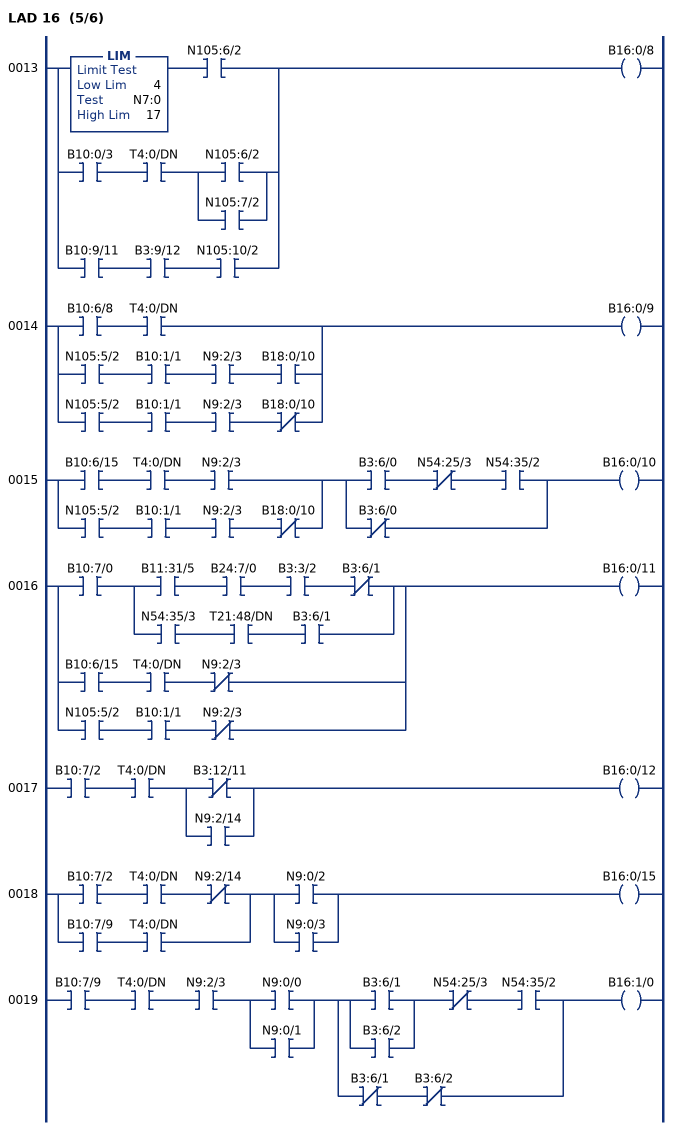
% Rung: 13 %
SOR BST LIM 4 N7:0 17 XIC N105:6/2 NXB XIC B10:0/3 XIC T4:0/DN BST XIC N105:6/2 NXB XIC N105:7/2 BND NXB XIC B10:9/11 XIC B3:9/12 XIC N105:10/2 BND OTE B16:0/8 EOR
% Rung: 14 %
SOR BST XIC B10:6/8 XIC T4:0/DN NXB XIC N105:5/2 XIC B10:1/1 XIC N9:2/3 XIC B18:0/10 NXB XIC N105:5/2 XIC B10:1/1 XIC N9:2/3 XIO B18:0/10 BND OTE B16:0/9 EOR
% Rung: 15 %
SOR BST XIC B10:6/15 XIC T4:0/DN XIC N9:2/3 NXB XIC N105:5/2 XIC B10:1/1 XIC N9:2/3 XIO B18:0/10 BND BST XIC B3:6/0 XIO N54:25/3 XIC N54:35/2 NXB XIO B3:6/0 BND OTE B16:0/10 EOR
% Rung: 16 %
SOR BST BST XIC B10:7/0 BST XIC B11:31/5 XIC B24:7/0 XIC B3:3/2 XIO B3:6/1 NXB XIC N54:35/3 XIC T21:48/DN XIC B3:6/1 BND NXB XIC B10:6/15 XIC T4:0/DN XIO N9:2/3 BND NXB XIC N105:5/2 XIC B10:1/1 XIO N9:2/3 BND OTE B16:0/11 EOR
% Rung: 17 %
SOR XIC B10:7/2 XIC T4:0/DN BST XIO B3:12/11 NXB XIC N9:2/14 BND OTE B16:0/12 EOR
% Rung: 18 %
SOR BST XIC B10:7/2 XIC T4:0/DN XIO N9:2/14 NXB XIC B10:7/9 XIC T4:0/DN BND BST XIC N9:0/2 NXB XIC N9:0/3 BND OTE B16:0/15 EOR
% Rung: 19 %
SOR XIC B10:7/9 XIC T4:0/DN XIC N9:2/3 BST XIC N9:0/0 NXB XIC N9:0/1 BND BST BST XIC B3:6/1 NXB XIC B3:6/2 BND XIO N54:25/3 XIC N54:35/2 NXB XIO B3:6/1 XIO B3:6/2 BND OTE B16:1/0 EOR

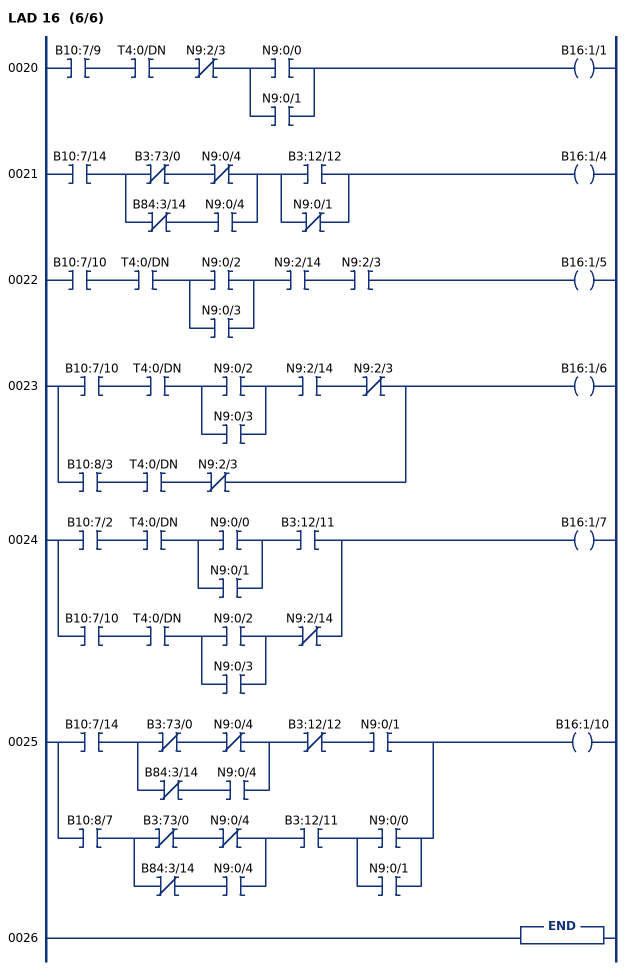
% Rung: 20 %
SOR XIC B10:7/9 XIC T4:0/DN XIO N9:2/3 BST XIC N9:0/0 NXB XIC N9:0/1 BND OTE B16:1/1 EOR
% Rung: 21 %
SOR XIC B10:7/14 BST XIO B3:73/0 XIO N9:0/4 NXB XIO B84:3/14 XIC N9:0/4 BND BST XIC B3:12/12 NXB XIO N9:0/1 BND OTE B16:1/4 EOR
% Rung: 22 %
SOR XIC B10:7/10 XIC T4:0/DN BST XIC N9:0/2 NXB XIC N9:0/3 BND XIC N9:2/14 XIC N9:2/3 OTE B16:1/5 EOR
% Rung: 23 %
SOR BST XIC B10:7/10 XIC T4:0/DN BST XIC N9:0/2 NXB XIC N9:0/3 BND XIC N9:2/14 XIO N9:2/3 NXB XIC B10:8/3 XIC T4:0/DN XIO N9:2/3 BND OTE B16:1/6 EOR
% Rung: 24 %
SOR BST XIC B10:7/2 XIC T4:0/DN BST XIC N9:0/0 NXB XIC N9:0/1 BND XIC B3:12/11 NXB XIC B10:7/10 XIC T4:0/DN BST XIC N9:0/2 NXB XIC N9:0/3 BND XIO N9:2/14 BND OTE B16:1/7 EOR
% Rung: 25 %
SOR BST XIC B10:7/14 BST XIO B3:73/0 XIO N9:0/4 NXB XIO B84:3/14 XIC N9:0/4 BND XIO B3:12/12 XIC N9:0/1 NXB XIC B10:8/7 BST XIO B3:73/0 XIO N9:0/4 NXB XIO B84:3/14 XIC N9:0/4 BND XIC B3:12/11 BST XIC N9:0/0 NXB XIC N9:0/1 BND BND OTE B16:1/10 EOR
% Rung: 26 %
SOR END EOR

LADDER 17
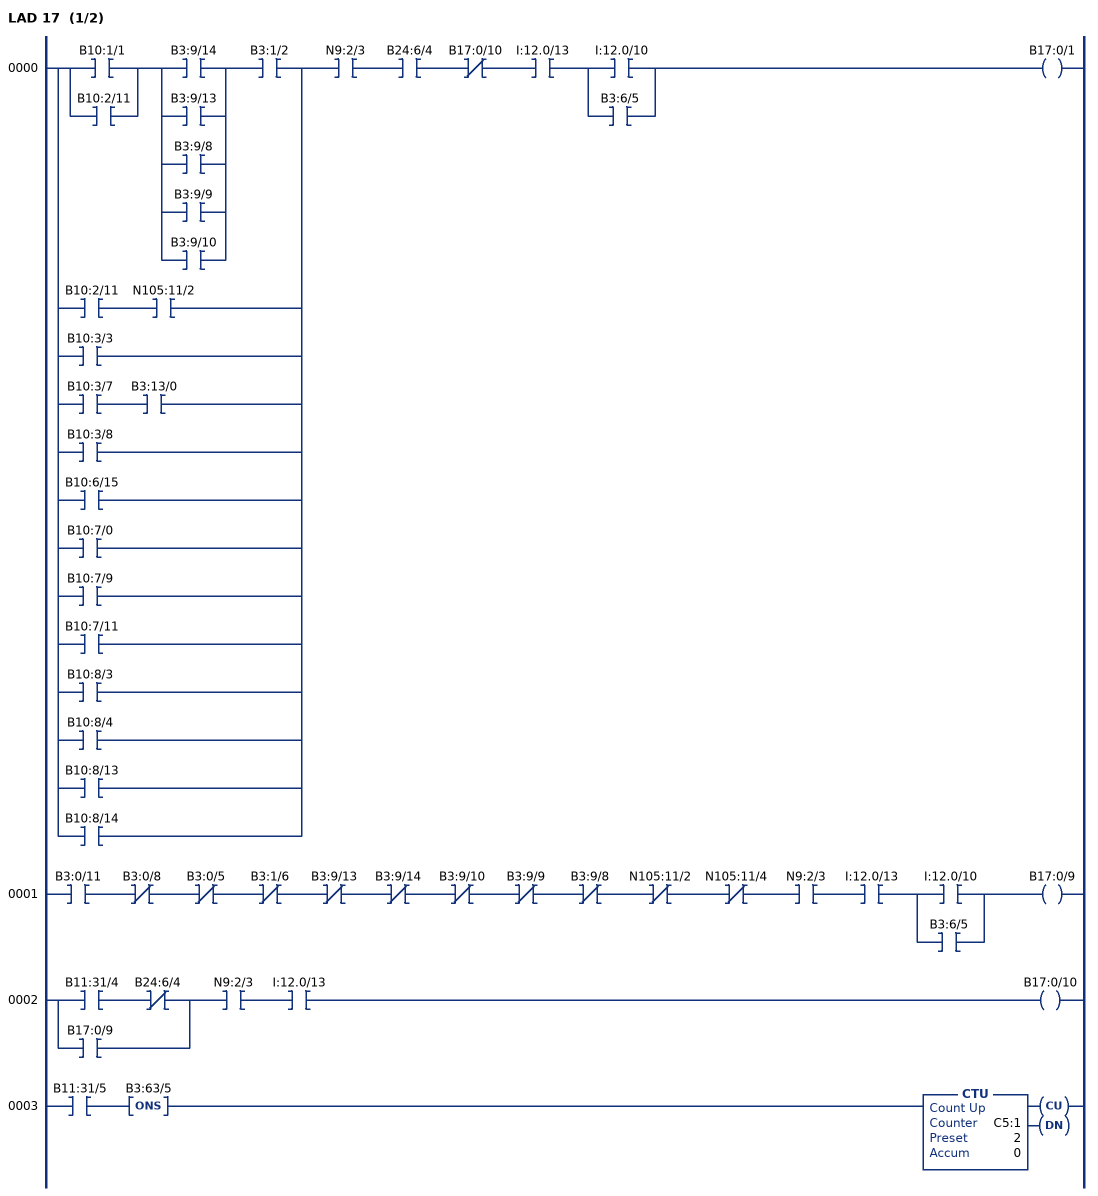
% Rung: 0 %
SOR BST BST XIC B10:1/1 NXB XIC B10:2/11 BND BST XIC B3:9/14 NXB XIC B3:9/13 NXB XIC B3:9/8 NXB XIC B3:9/9 NXB XIC B3:9/10 BND XIC B3:1/2 NXB XIC B10:2/11 XIC N105:11/2 NXB XIC B10:3/3 NXB XIC B10:3/7 XIC B3:13/0 NXB XIC B10:3/8 NXB XIC B10:6/15 NXB XIC B10:7/0 NXB XIC B10:7/9 NXB XIC B10:7/11 NXB XIC B10:8/3 NXB XIC B10:8/4 NXB XIC B10:8/13 NXB XIC B10:8/14 BND XIC N9:2/3 XIC B24:6/4 XIO B17:0/10 XIC I:12.0/13 BST XIC I:12.0/10 NXB XIC B3:6/5 BND OTE B17:0/1 EOR
% Rung: 1 %
SOR XIC B3:0/11 XIO B3:0/8 XIO B3:0/5 XIO B3:1/6 XIO B3:9/13 XIO B3:9/14 XIO B3:9/10 XIO B3:9/9 XIO B3:9/8 XIO N105:11/2 XIO N105:11/4 XIC N9:2/3 XIC I:12.0/13 BST XIC I:12.0/10 NXB XIC B3:6/5 BND OTE B17:0/9 EOR
% Rung: 2 %
SOR BST XIC B11:31/4 XIO B24:6/4 NXB XIC B17:0/9 BND XIC N9:2/3 XIC I:12.0/13 OTE B17:0/10 EOR
% Rung: 3 %
SOR XIC B11:31/5 OSR B3:63/5 CTU C5:1 2 0 EOR

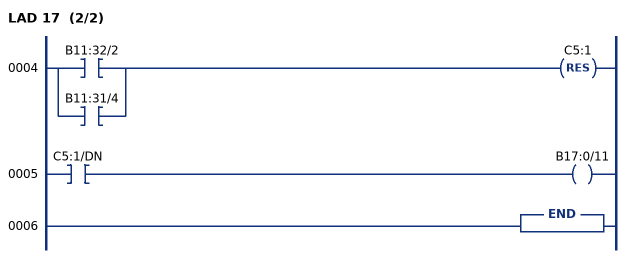
% Rung: 4 %
SOR BST XIC B11:32/2 NXB XIC B11:31/4 BND RES C5:1 EOR
% Rung: 5 %
SOR XIC C5:1/DN OTE B17:0/11 EOR
% Rung: 6 %
SOR END EOR

LADDER 18
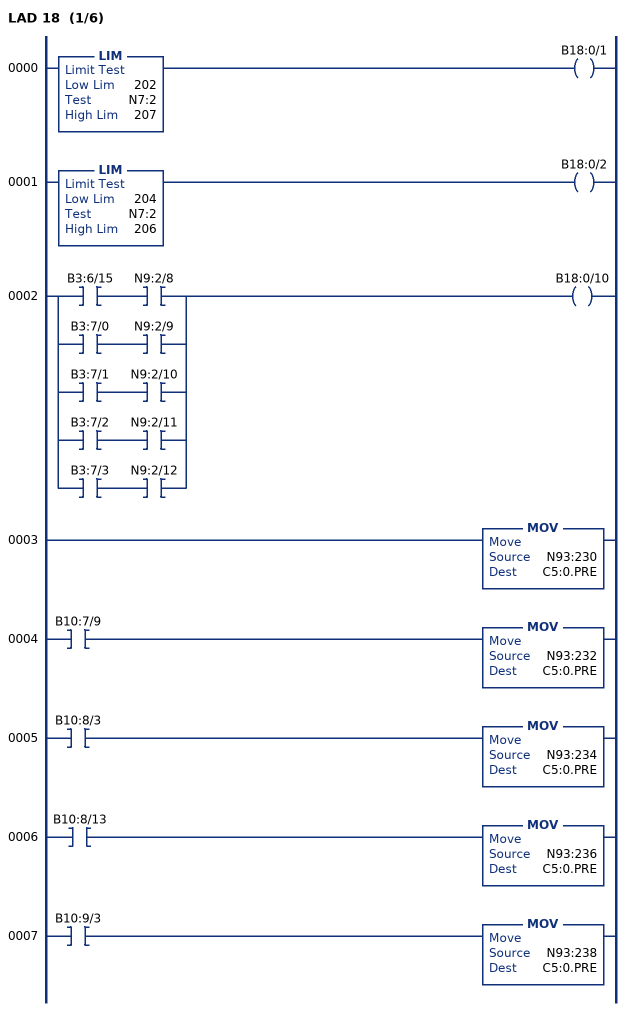
% Rung: 0 %
SOR LIM 202 N7:2 207 OTE B18:0/1 EOR
% Rung: 1 %
SOR LIM 204 N7:2 206 OTE B18:0/2 EOR
% Rung: 2 %
SOR BST XIC B3:6/15 XIC N9:2/8 NXB XIC B3:7/0 XIC N9:2/9 NXB XIC B3:7/1 XIC N9:2/10 NXB XIC B3:7/2 XIC N9:2/11 NXB XIC B3:7/3 XIC N9:2/12 BND OTE B18:0/10 EOR
% Rung: 3 %
SOR MOV N93:230 C5:0.PRE EOR
% Rung: 4 %
SOR XIC B10:7/9 MOV N93:232 C5:0.PRE EOR
% Rung: 5 %
SOR XIC B10:8/3 MOV N93:234 C5:0.PRE EOR
% Rung: 6 %
SOR XIC B10:8/13 MOV N93:236 C5:0.PRE EOR
% Rung: 7 %
SOR XIC B10:9/3 MOV N93:238 C5:0.PRE EOR

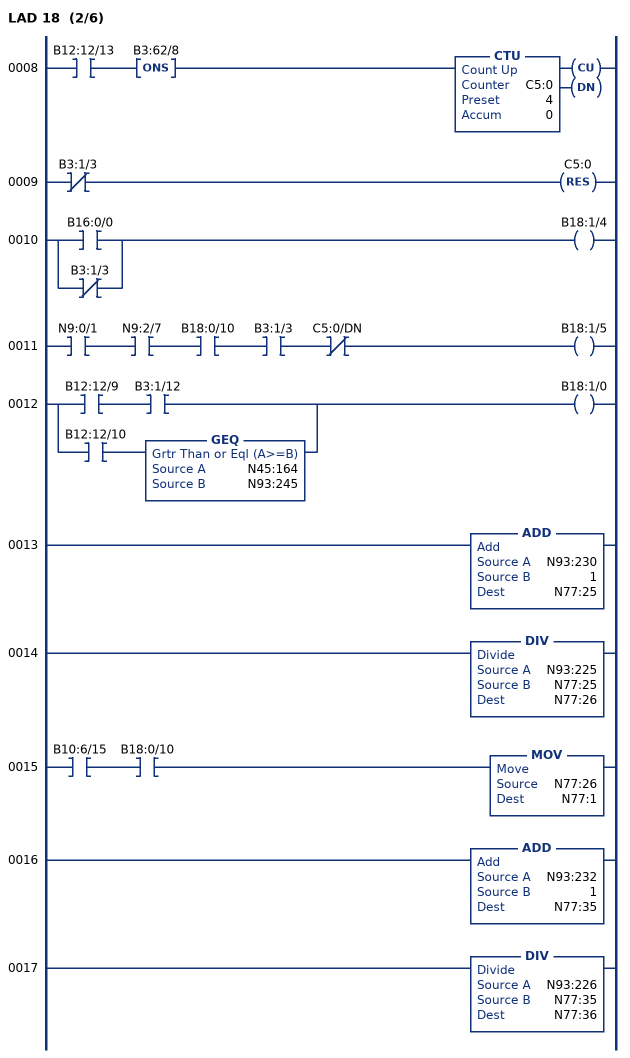
% Rung: 8 %
SOR XIC B12:12/13 OSR B3:62/8 CTU C5:0 4 0 EOR
% Rung: 9 %
SOR XIO B3:1/3 RES C5:0 EOR
% Rung: 10 %
SOR BST XIC B16:0/0 NXB XIO B3:1/3 BND OTE B18:1/4 EOR
% Rung: 11 %
SOR XIC N9:0/1 XIC N9:2/7 XIC B18:0/10 XIC B3:1/3 XIO C5:0/DN OTE B18:1/5 EOR
% Rung: 12 %
SOR BST XIC B12:12/9 XIC B3:1/12 NXB XIC B12:12/10 GEQ N45:164 N93:245 BND OTE B18:1/0 EOR
% Rung: 13 %
SOR ADD N93:230 1 N77:25 EOR
% Rung: 14 %
SOR DIV N93:225 N77:25 N77:26 EOR
% Rung: 15 %
SOR XIC B10:6/15 XIC B18:0/10 MOV N77:26 N77:1 EOR
% Rung: 16 %
SOR ADD N93:232 1 N77:35 EOR
% Rung: 17 %
SOR DIV N93:226 N77:35 N77:36 EOR

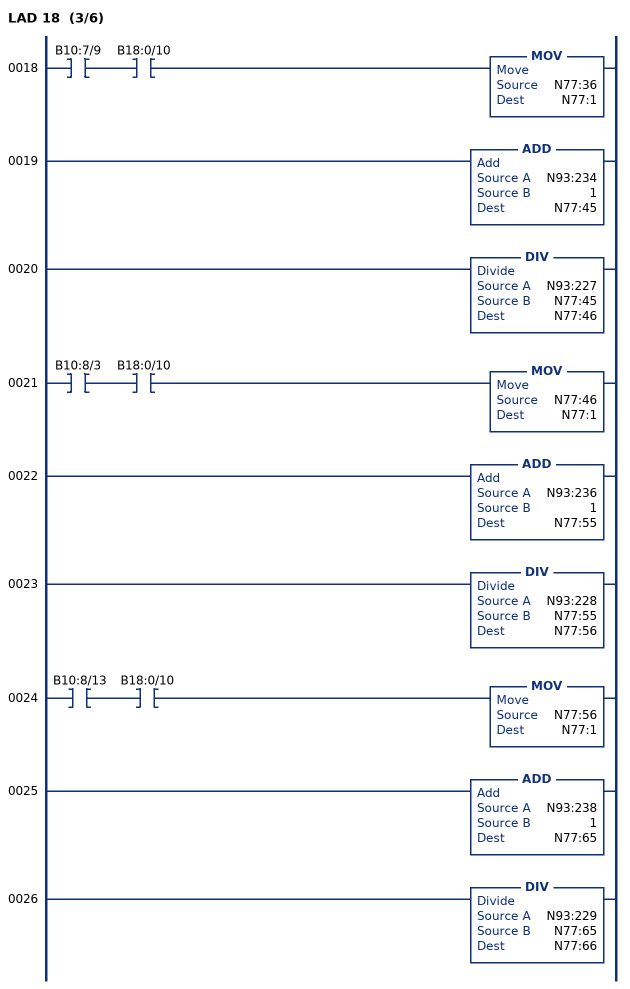
% Rung: 18 %
SOR XIC B10:7/9 XIC B18:0/10 MOV N77:36 N77:1 EOR
% Rung: 19 %
SOR ADD N93:234 1 N77:45 EOR
% Rung: 20 %
SOR DIV N93:227 N77:45 N77:46 EOR
% Rung: 21 %
SOR XIC B10:8/3 XIC B18:0/10 MOV N77:46 N77:1 EOR
% Rung: 22 %
SOR ADD N93:236 1 N77:55 EOR
% Rung: 23 %
SOR DIV N93:228 N77:55 N77:56 EOR
% Rung: 24 %
SOR XIC B10:8/13 XIC B18:0/10 MOV N77:56 N77:1 EOR
% Rung: 25 %
SOR ADD N93:238 1 N77:65 EOR
% Rung: 26 %
SOR DIV N93:229 N77:65 N77:66 EOR

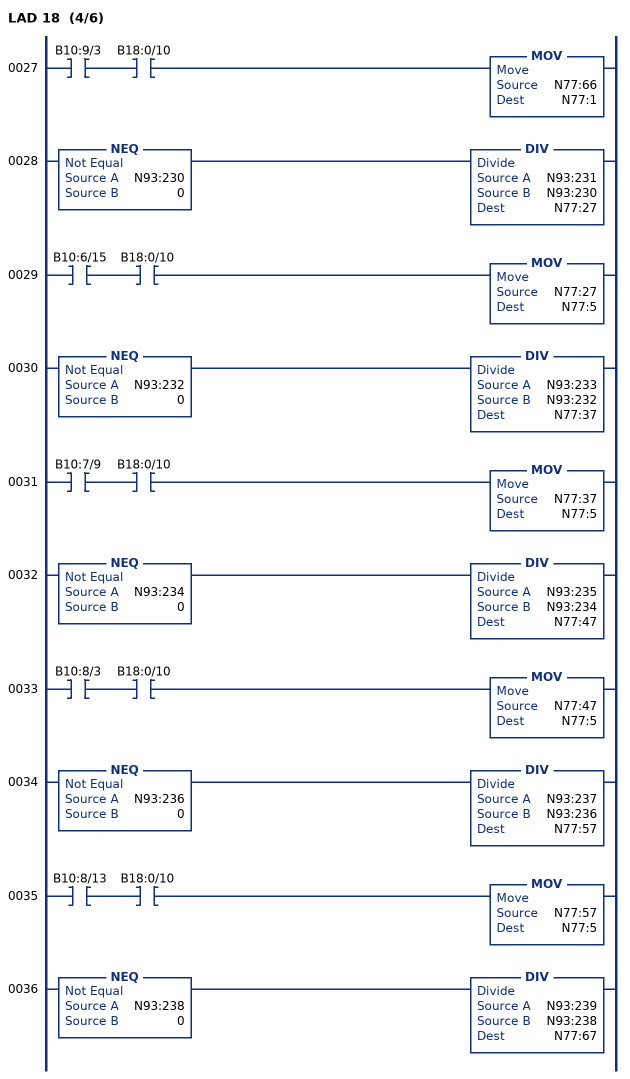
% Rung: 27 %
SOR XIC B10:9/3 XIC B18:0/10 MOV N77:66 N77:1 EOR
% Rung: 28 %
SOR NEQ N93:230 0 DIV N93:231 N93:230 N77:27 EOR
% Rung: 29 %
SOR XIC B10:6/15 XIC B18:0/10 MOV N77:27 N77:5 EOR
% Rung: 30 %
SOR NEQ N93:232 0 DIV N93:233 N93:232 N77:37 EOR
% Rung: 31 %
SOR XIC B10:7/9 XIC B18:0/10 MOV N77:37 N77:5 EOR
% Rung: 32 %
SOR NEQ N93:234 0 DIV N93:235 N93:234 N77:47 EOR
% Rung: 33 %
SOR XIC B10:8/3 XIC B18:0/10 MOV N77:47 N77:5 EOR
% Rung: 34 %
SOR NEQ N93:236 0 DIV N93:237 N93:236 N77:57 EOR
% Rung: 35 %
SOR XIC B10:8/13 XIC B18:0/10 MOV N77:57 N77:5 EOR
% Rung: 36 %
SOR NEQ N93:238 0 DIV N93:239 N93:238 N77:67 EOR

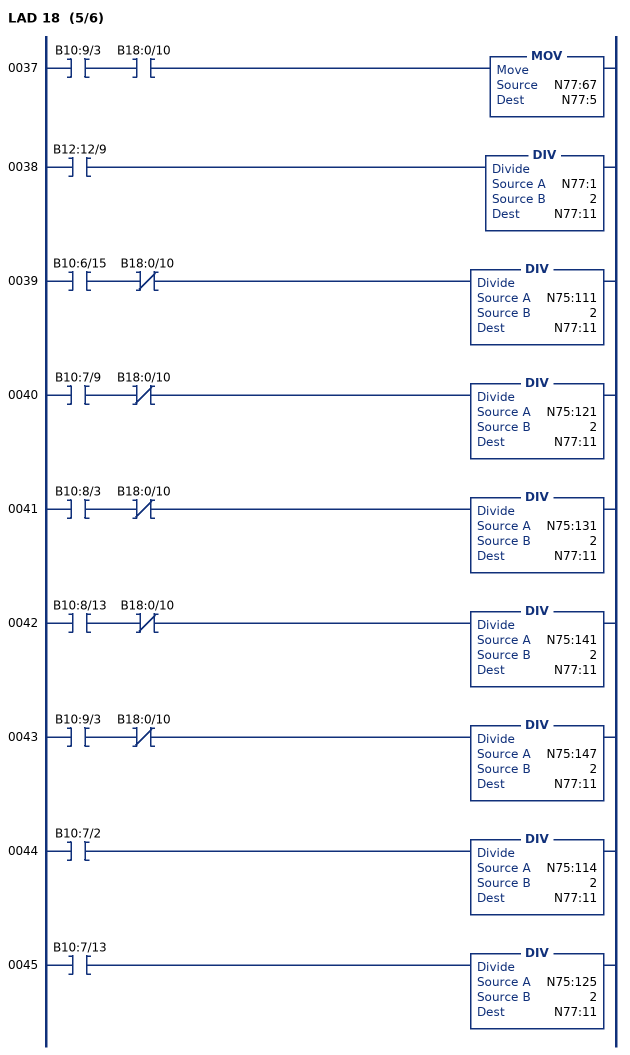
% Rung: 37 %
SOR XIC B10:9/3 XIC B18:0/10 MOV N77:67 N77:5 EOR
% Rung: 38 %
SOR XIC B12:12/9 DIV N77:1 2 N77:11 EOR
% Rung: 39 %
SOR XIC B10:6/15 XIO B18:0/10 DIV N75:111 2 N77:11 EOR
% Rung: 40 %
SOR XIC B10:7/9 XIO B18:0/10 DIV N75:121 2 N77:11 EOR
% Rung: 41 %
SOR XIC B10:8/3 XIO B18:0/10 DIV N75:131 2 N77:11 EOR
% Rung: 42 %
SOR XIC B10:8/13 XIO B18:0/10 DIV N75:141 2 N77:11 EOR
% Rung: 43 %
SOR XIC B10:9/3 XIO B18:0/10 DIV N75:147 2 N77:11 EOR
% Rung: 44 %
SOR XIC B10:7/2 DIV N75:114 2 N77:11 EOR
% Rung: 45 %
SOR XIC B10:7/13 DIV N75:125 2 N77:11 EOR

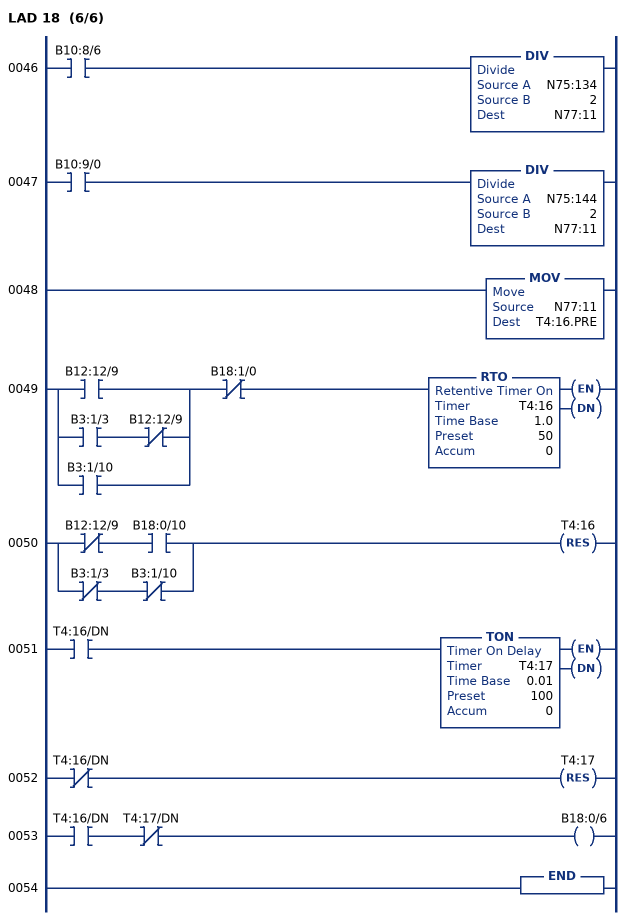
% Rung: 46 %
SOR XIC B10:8/6 DIV N75:134 2 N77:11 EOR
% Rung: 47 %
SOR XIC B10:9/0 DIV N75:144 2 N77:11 EOR
% Rung: 48 %
SOR MOV N77:11 T4:16.PRE EOR
% Rung: 49 %
SOR BST XIC B12:12/9 NXB XIC B3:1/3 XIO B12:12/9 NXB XIC B3:1/10 BND XIO B18:1/0 RTO T4:16 1.0 50 0 EOR
% Rung: 50 %
SOR BST XIO B12:12/9 XIC B18:0/10 NXB XIO B3:1/3 XIO B3:1/10 BND RES T4:16 EOR
% Rung: 51 %
SOR XIC T4:16/DN TON T4:17 0.01 100 0 EOR
% Rung: 52 %
SOR XIO T4:16/DN RES T4:17 EOR
% Rung: 53 %
SOR XIC T4:16/DN XIO T4:17/DN OTE B18:0/6 EOR
% Rung: 54 %
SOR END EOR

LADDER 21
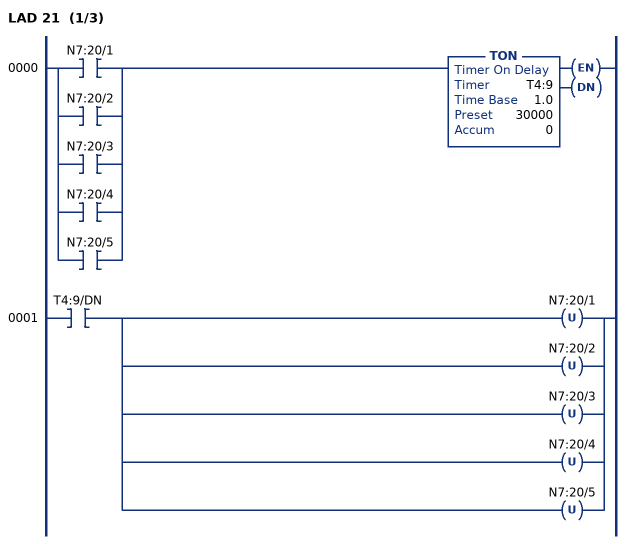
% Rung: 0 %
SOR BST XIC N7:20/1 NXB XIC N7:20/2 NXB XIC N7:20/3 NXB XIC N7:20/4 NXB XIC N7:20/5 BND TON T4:9 1.0 30000 0 EOR
% Rung: 1 %
SOR XIC T4:9/DN BST OTU N7:20/1 NXB OTU N7:20/2 NXB OTU N7:20/3 NXB OTU N7:20/4 NXB OTU N7:20/5 BND EOR

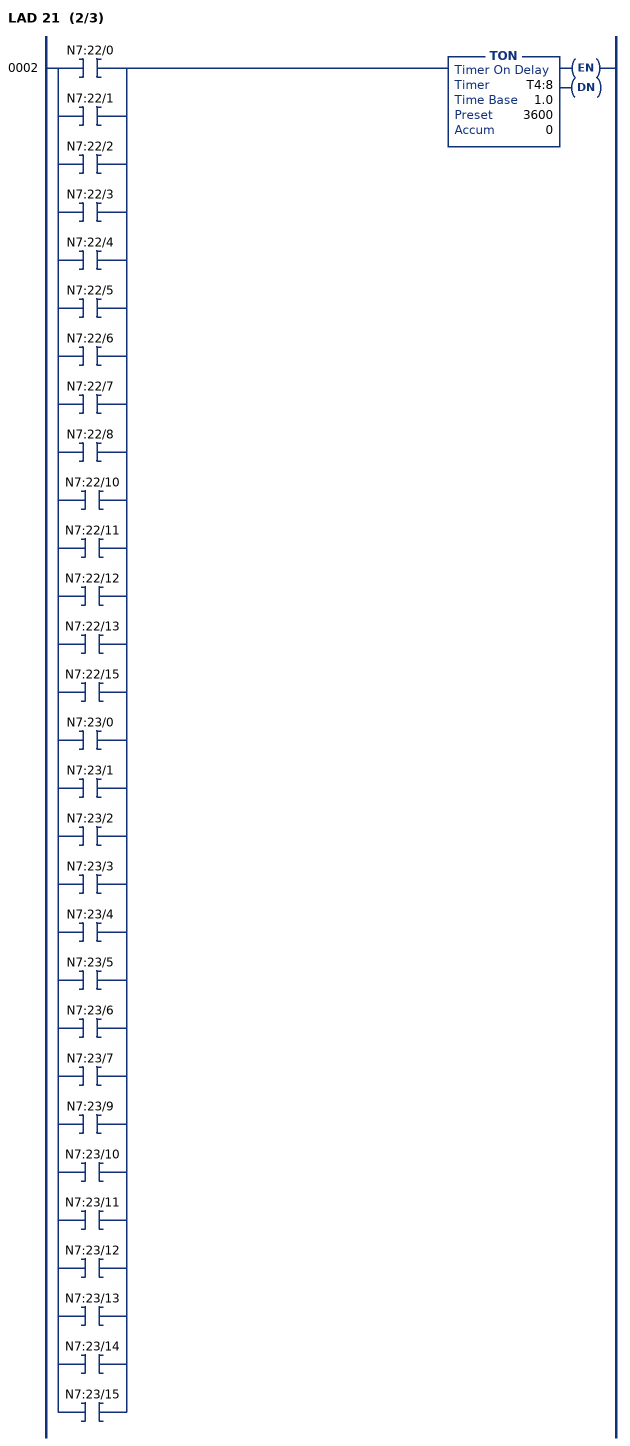
% Rung: 2 %
SOR BST XIC N7:22/0 NXB XIC N7:22/1 NXB XIC N7:22/2 NXB XIC N7:22/3 NXB XIC N7:22/4 NXB XIC N7:22/5 NXB XIC N7:22/6 NXB XIC N7:22/7 NXB XIC N7:22/8 NXB XIC N7:22/10 NXB XIC N7:22/11 NXB XIC N7:22/12 NXB XIC N7:22/13 NXB XIC N7:22/15 NXB XIC N7:23/0 NXB XIC N7:23/1 NXB XIC N7:23/2 NXB XIC N7:23/3 NXB XIC N7:23/4 NXB XIC N7:23/5 NXB XIC N7:23/6 NXB XIC N7:23/7 NXB XIC N7:23/9 NXB XIC N7:23/10 NXB XIC N7:23/11 NXB XIC N7:23/12 NXB XIC N7:23/13 NXB XIC N7:23/14 NXB XIC N7:23/15 BND TON T4:8 1.0 3600 0 EOR

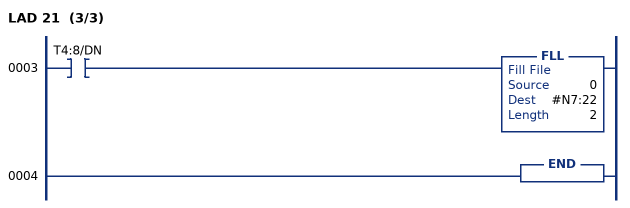
% Rung: 3 %
SOR XIC T4:8/DN FLL 0 #N7:22 2 EOR
% Rung: 4 %
SOR END EOR

LADDER 22
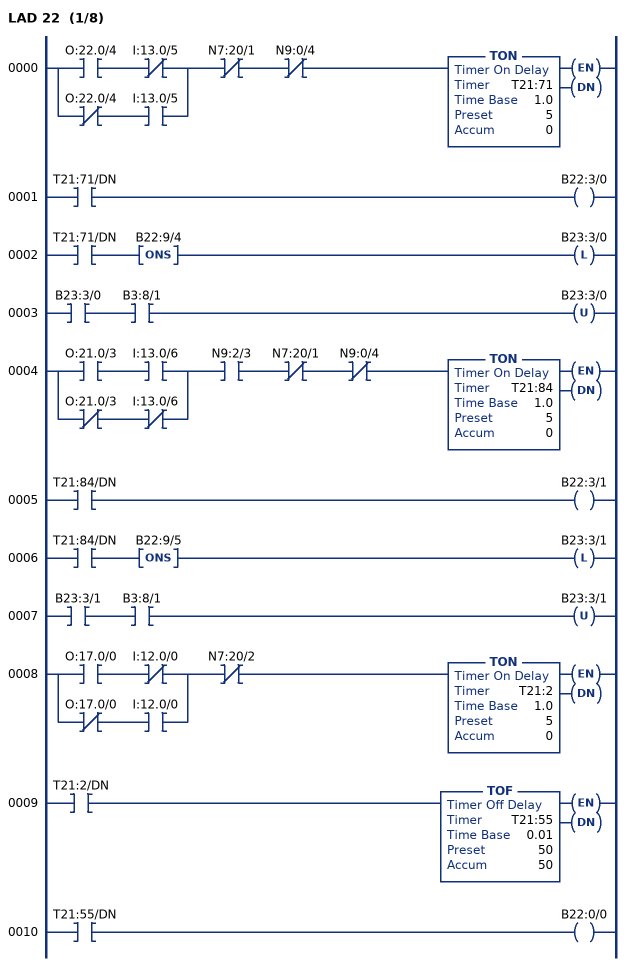
% Rung: 0 %
SOR BST XIC O:22.0/4 XIO I:13.0/5 NXB XIO O:22.0/4 XIC I:13.0/5 BND XIO N7:20/1 XIO N9:0/4 TON T21:71 1.0 5 0 EOR
% Rung: 1 %
SOR XIC T21:71/DN OTE B22:3/0 EOR
% Rung: 2 %
SOR XIC T21:71/DN OSR B22:9/4 OTL B23:3/0 EOR
% Rung: 3 %
SOR XIC B23:3/0 XIC B3:8/1 OTU B23:3/0 EOR
% Rung: 4 %
SOR BST XIC O:21.0/3 XIC I:13.0/6 NXB XIO O:21.0/3 XIO I:13.0/6 BND XIC N9:2/3 XIO N7:20/1 XIO N9:0/4 TON T21:84 1.0 5 0 EOR
% Rung: 5 %
SOR XIC T21:84/DN OTE B22:3/1 EOR
% Rung: 6 %
SOR XIC T21:84/DN OSR B22:9/5 OTL B23:3/1 EOR
% Rung: 7 %
SOR XIC B23:3/1 XIC B3:8/1 OTU B23:3/1 EOR
% Rung: 8 %
SOR BST XIC O:17.0/0 XIO I:12.0/0 NXB XIO O:17.0/0 XIC I:12.0/0 BND XIO N7:20/2 TON T21:2 1.0 5 0 EOR
% Rung: 9 %
SOR XIC T21:2/DN TOF T21:55 0.01 50 50 EOR
% Rung: 10 %
SOR XIC T21:55/DN OTE B22:0/0 EOR

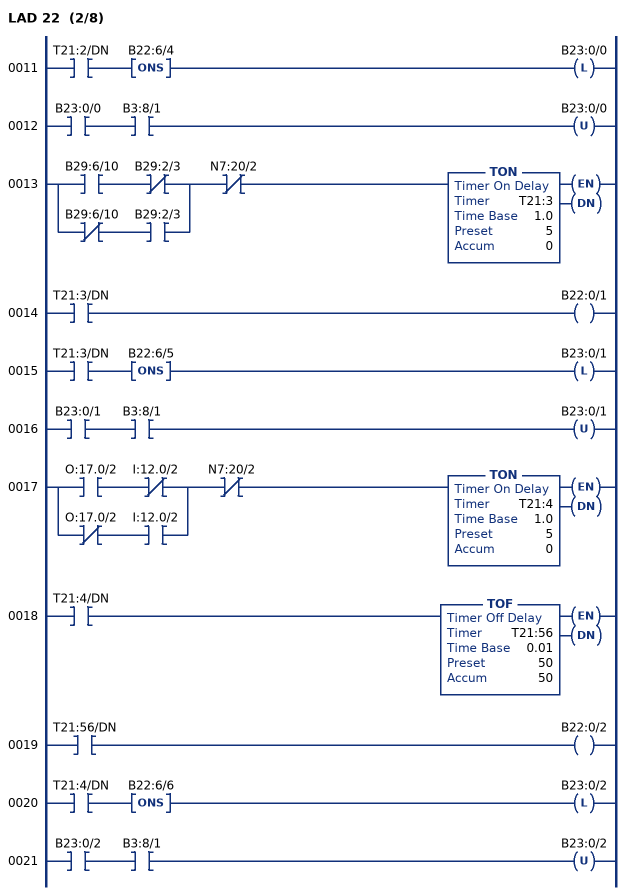
% Rung: 11 %
SOR XIC T21:2/DN OSR B22:6/4 OTL B23:0/0 EOR
% Rung: 12 %
SOR XIC B23:0/0 XIC B3:8/1 OTU B23:0/0 EOR
% Rung: 13 %
SOR BST XIC B29:6/10 XIO B29:2/3 NXB XIO B29:6/10 XIC B29:2/3 BND XIO N7:20/2 TON T21:3 1.0 5 0 EOR
% Rung: 14 %
SOR XIC T21:3/DN OTE B22:0/1 EOR
% Rung: 15 %
SOR XIC T21:3/DN OSR B22:6/5 OTL B23:0/1 EOR
% Rung: 16 %
SOR XIC B23:0/1 XIC B3:8/1 OTU B23:0/1 EOR
% Rung: 17 %
SOR BST XIC O:17.0/2 XIO I:12.0/2 NXB XIO O:17.0/2 XIC I:12.0/2 BND XIO N7:20/2 TON T21:4 1.0 5 0 EOR
% Rung: 18 %
SOR XIC T21:4/DN TOF T21:56 0.01 50 50 EOR
% Rung: 19 %
SOR XIC T21:56/DN OTE B22:0/2 EOR
% Rung: 20 %
SOR XIC T21:4/DN OSR B22:6/6 OTL B23:0/2 EOR
% Rung: 21 %
SOR XIC B23:0/2 XIC B3:8/1 OTU B23:0/2 EOR

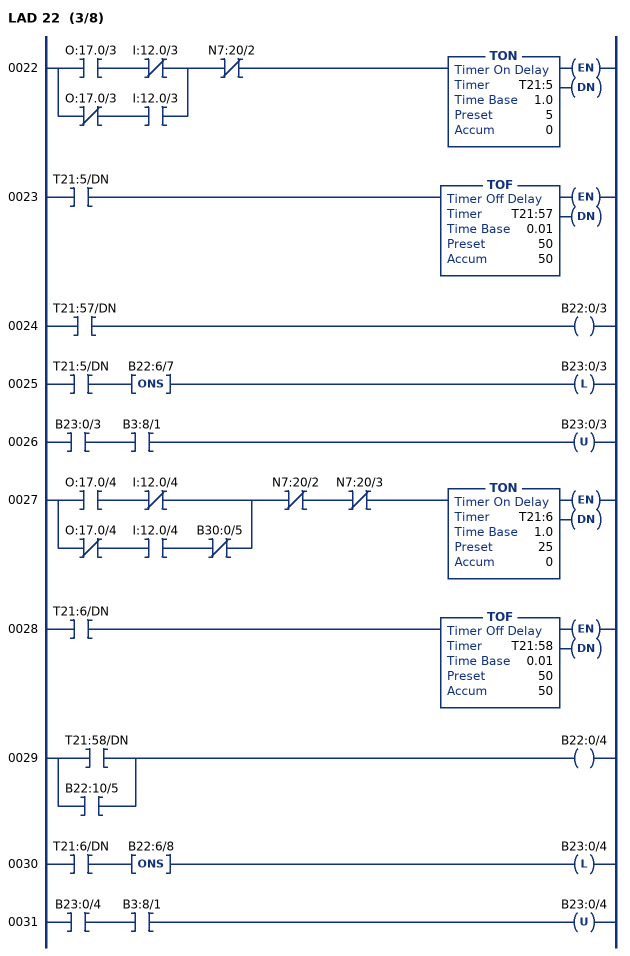
% Rung: 22 %
SOR BST XIC O:17.0/3 XIO I:12.0/3 NXB XIO O:17.0/3 XIC I:12.0/3 BND XIO N7:20/2 TON T21:5 1.0 5 0 EOR
% Rung: 23 %
SOR XIC T21:5/DN TOF T21:57 0.01 50 50 EOR
% Rung: 24 %
SOR XIC T21:57/DN OTE B22:0/3 EOR
% Rung: 25 %
SOR XIC T21:5/DN OSR B22:6/7 OTL B23:0/3 EOR
% Rung: 26 %
SOR XIC B23:0/3 XIC B3:8/1 OTU B23:0/3 EOR
% Rung: 27 %
SOR BST XIC O:17.0/4 XIO I:12.0/4 NXB XIO O:17.0/4 XIC I:12.0/4 XIO B30:0/5 BND XIO N7:20/2 XIO N7:20/3 TON T21:6 1.0 25 0 EOR
% Rung: 28 %
SOR XIC T21:6/DN TOF T21:58 0.01 50 50 EOR
% Rung: 29 %
SOR BST XIC T21:58/DN NXB XIC B22:10/5 BND OTE B22:0/4 EOR
% Rung: 30 %
SOR XIC T21:6/DN OSR B22:6/8 OTL B23:0/4 EOR
% Rung: 31 %
SOR XIC B23:0/4 XIC B3:8/1 OTU B23:0/4 EOR

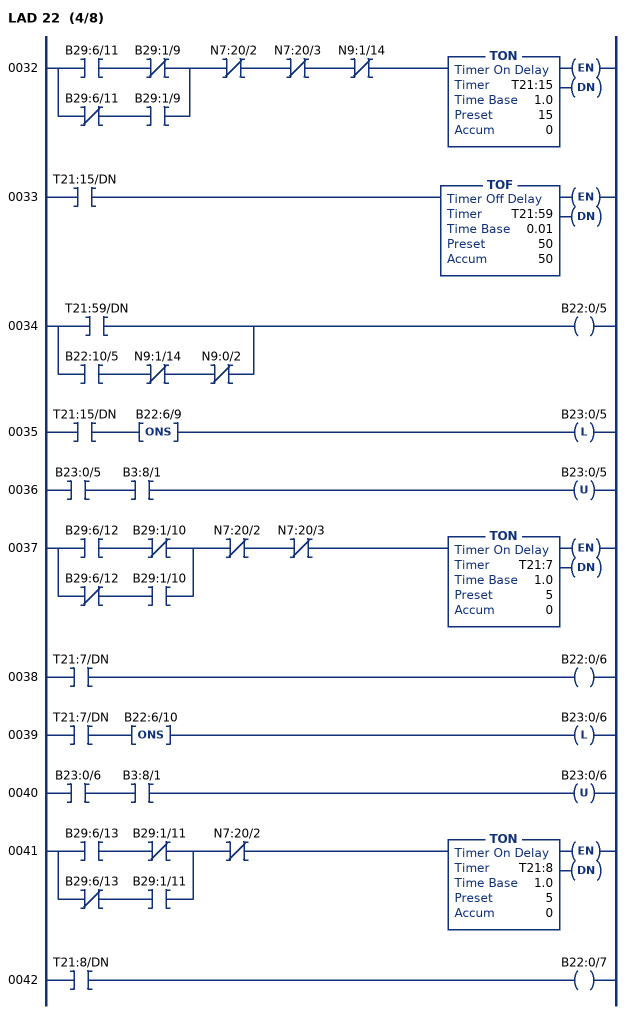
% Rung: 32 %
SOR BST XIC B29:6/11 XIO B29:1/9 NXB XIO B29:6/11 XIC B29:1/9 BND XIO N7:20/2 XIO N7:20/3 XIO N9:1/14 TON T21:15 1.0 15 0 EOR
% Rung: 33 %
SOR XIC T21:15/DN TOF T21:59 0.01 50 50 EOR
% Rung: 34 %
SOR BST XIC T21:59/DN NXB XIC B22:10/5 XIO N9:1/14 XIO N9:0/2 BND OTE B22:0/5 EOR
% Rung: 35 %
SOR XIC T21:15/DN OSR B22:6/9 OTL B23:0/5 EOR
% Rung: 36 %
SOR XIC B23:0/5 XIC B3:8/1 OTU B23:0/5 EOR
% Rung: 37 %
SOR BST XIC B29:6/12 XIO B29:1/10 NXB XIO B29:6/12 XIC B29:1/10 BND XIO N7:20/2 XIO N7:20/3 TON T21:7 1.0 5 0 EOR
% Rung: 38 %
SOR XIC T21:7/DN OTE B22:0/6 EOR
% Rung: 39 %
SOR XIC T21:7/DN OSR B22:6/10 OTL B23:0/6 EOR
% Rung: 40 %
SOR XIC B23:0/6 XIC B3:8/1 OTU B23:0/6 EOR
% Rung: 41 %
SOR BST XIC B29:6/13 XIO B29:1/11 NXB XIO B29:6/13 XIC B29:1/11 BND XIO N7:20/2 TON T21:8 1.0 5 0 EOR
% Rung: 42 %
SOR XIC T21:8/DN OTE B22:0/7 EOR

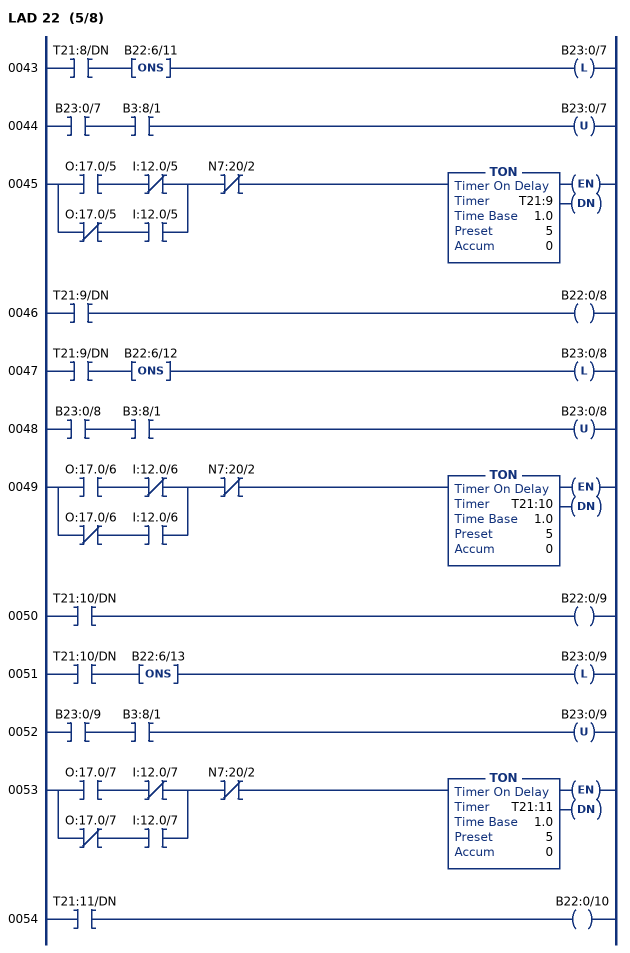
% Rung: 43 %
SOR XIC T21:8/DN OSR B22:6/11 OTL B23:0/7 EOR
% Rung: 44 %
SOR XIC B23:0/7 XIC B3:8/1 OTU B23:0/7 EOR
% Rung: 45 %
SOR BST XIC O:17.0/5 XIO I:12.0/5 NXB XIO O:17.0/5 XIC I:12.0/5 BND XIO N7:20/2 TON T21:9 1.0 5 0 EOR
% Rung: 46 %
SOR XIC T21:9/DN OTE B22:0/8 EOR
% Rung: 47 %
SOR XIC T21:9/DN OSR B22:6/12 OTL B23:0/8 EOR
% Rung: 48 %
SOR XIC B23:0/8 XIC B3:8/1 OTU B23:0/8 EOR
% Rung: 49 %
SOR BST XIC O:17.0/6 XIO I:12.0/6 NXB XIO O:17.0/6 XIC I:12.0/6 BND XIO N7:20/2 TON T21:10 1.0 5 0 EOR
% Rung: 50 %
SOR XIC T21:10/DN OTE B22:0/9 EOR
% Rung: 51 %
SOR XIC T21:10/DN OSR B22:6/13 OTL B23:0/9 EOR
% Rung: 52 %
SOR XIC B23:0/9 XIC B3:8/1 OTU B23:0/9 EOR
% Rung: 53 %
SOR BST XIC O:17.0/7 XIO I:12.0/7 NXB XIO O:17.0/7 XIC I:12.0/7 BND XIO N7:20/2 TON T21:11 1.0 5 0 EOR
% Rung: 54 %
SOR XIC T21:11/DN OTE B22:0/10 EOR

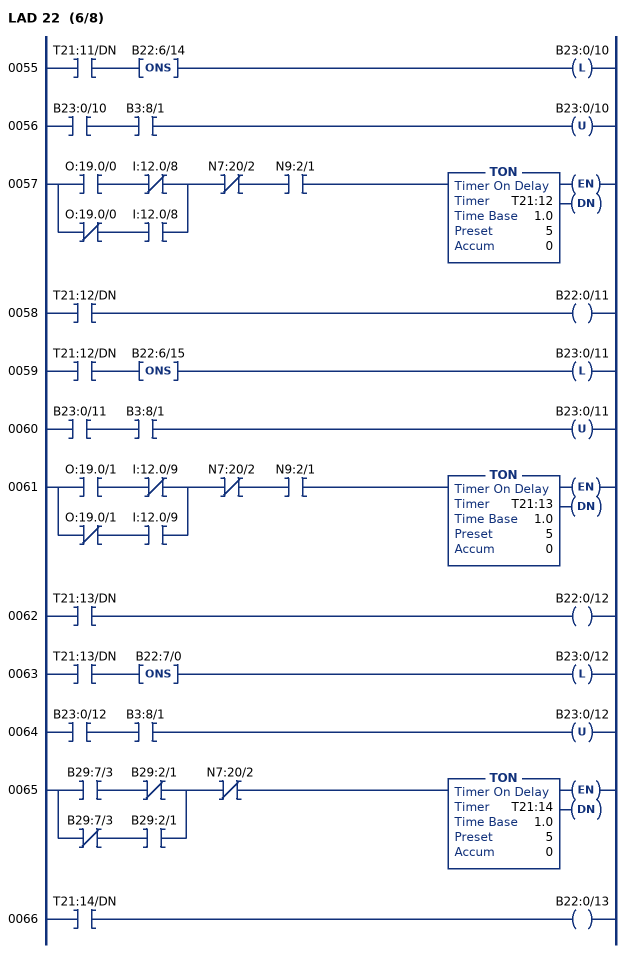
% Rung: 55 %
SOR XIC T21:11/DN OSR B22:6/14 OTL B23:0/10 EOR
% Rung: 56 %
SOR XIC B23:0/10 XIC B3:8/1 OTU B23:0/10 EOR
% Rung: 57 %
SOR BST XIC O:19.0/0 XIO I:12.0/8 NXB XIO O:19.0/0 XIC I:12.0/8 BND XIO N7:20/2 XIC N9:2/1 TON T21:12 1.0 5 0 EOR
% Rung: 58 %
SOR XIC T21:12/DN OTE B22:0/11 EOR
% Rung: 59 %
SOR XIC T21:12/DN OSR B22:6/15 OTL B23:0/11 EOR
% Rung: 60 %
SOR XIC B23:0/11 XIC B3:8/1 OTU B23:0/11 EOR
% Rung: 61 %
SOR BST XIC O:19.0/1 XIO I:12.0/9 NXB XIO O:19.0/1 XIC I:12.0/9 BND XIO N7:20/2 XIC N9:2/1 TON T21:13 1.0 5 0 EOR
% Rung: 62 %
SOR XIC T21:13/DN OTE B22:0/12 EOR
% Rung: 63 %
SOR XIC T21:13/DN OSR B22:7/0 OTL B23:0/12 EOR
% Rung: 64 %
SOR XIC B23:0/12 XIC B3:8/1 OTU B23:0/12 EOR
% Rung: 65 %
SOR BST XIC B29:7/3 XIO B29:2/1 NXB XIO B29:7/3 XIC B29:2/1 BND XIO N7:20/2 TON T21:14 1.0 5 0 EOR
% Rung: 66 %
SOR XIC T21:14/DN OTE B22:0/13 EOR

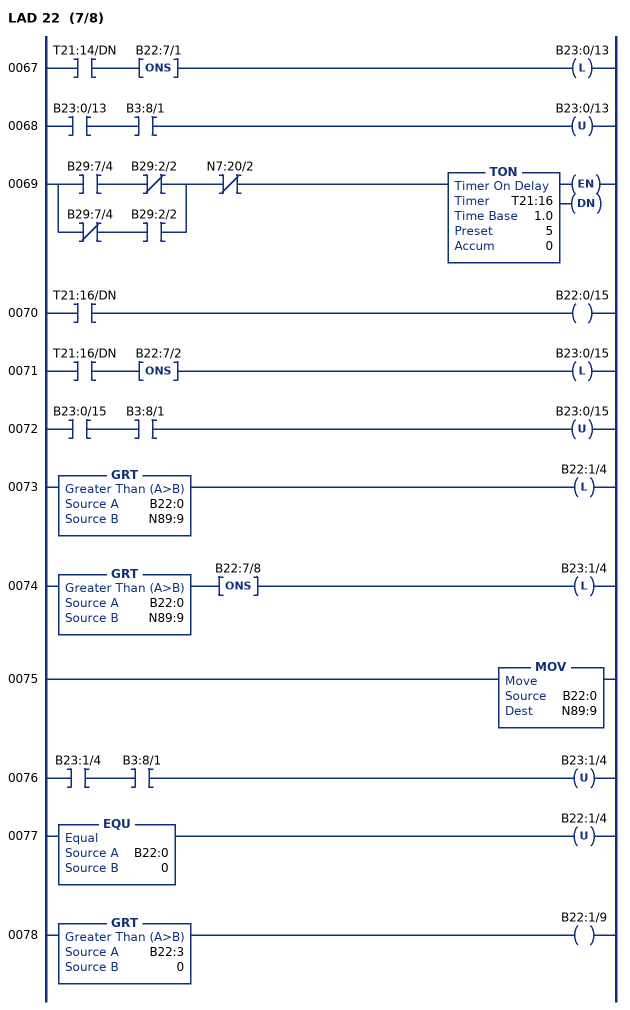
% Rung: 67 %
SOR XIC T21:14/DN OSR B22:7/1 OTL B23:0/13 EOR
% Rung: 68 %
SOR XIC B23:0/13 XIC B3:8/1 OTU B23:0/13 EOR
% Rung: 69 %
SOR BST XIC B29:7/4 XIO B29:2/2 NXB XIO B29:7/4 XIC B29:2/2 BND XIO N7:20/2 TON T21:16 1.0 5 0 EOR
% Rung: 70 %
SOR XIC T21:16/DN OTE B22:0/15 EOR
% Rung: 71 %
SOR XIC T21:16/DN OSR B22:7/2 OTL B23:0/15 EOR
% Rung: 72 %
SOR XIC B23:0/15 XIC B3:8/1 OTU B23:0/15 EOR
% Rung: 73 %
SOR GRT B22:0 N89:9 OTL B22:1/4 EOR
% Rung: 74 %
SOR GRT B22:0 N89:9 OSR B22:7/8 OTL B23:1/4 EOR
% Rung: 75 %
SOR MOV B22:0 N89:9 EOR
% Rung: 76 %
SOR XIC B23:1/4 XIC B3:8/1 OTU B23:1/4 EOR
% Rung: 77 %
SOR EQU B22:0 0 OTU B22:1/4 EOR
% Rung: 78 %
SOR GRT B22:3 0 OTE B22:1/9 EOR

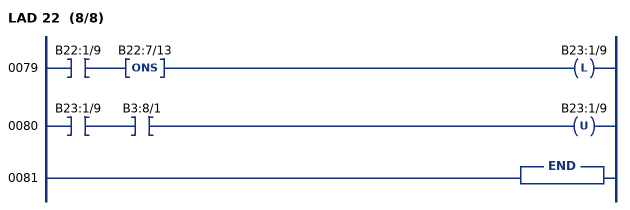
% Rung: 79 %
SOR XIC B22:1/9 OSR B22:7/13 OTL B23:1/9 EOR
% Rung: 80 %
SOR XIC B23:1/9 XIC B3:8/1 OTU B23:1/9 EOR
% Rung: 81 %
SOR END EOR

LADDER 23
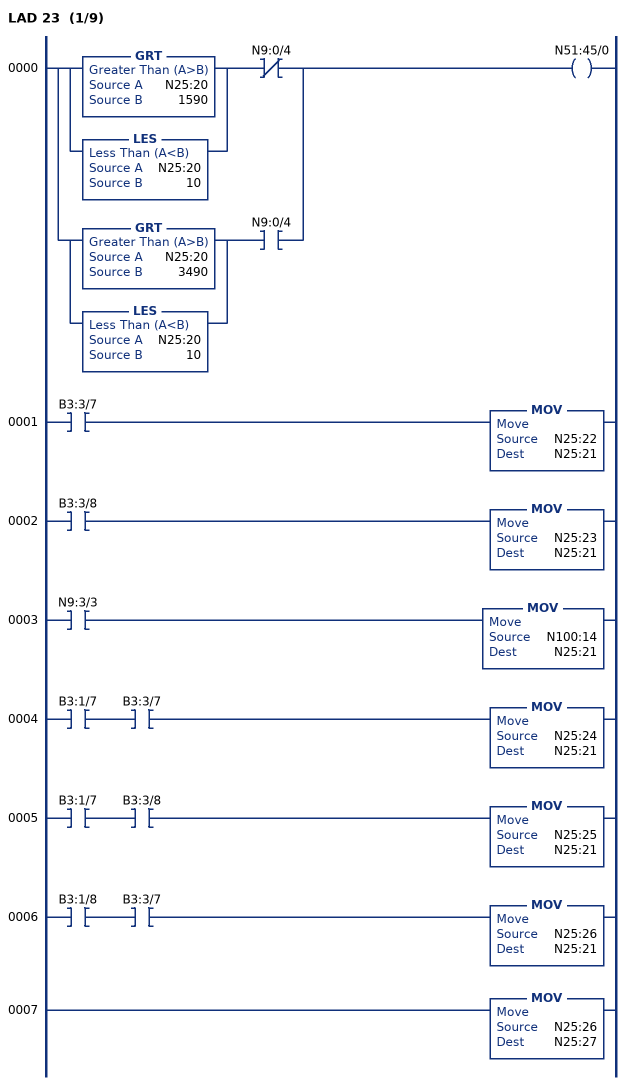
% Rung: 0 %
SOR BST BST GRT N25:20 1590 NXB LES N25:20 10 BND XIO N9:0/4 NXB BST GRT N25:20 3490 NXB LES N25:20 10 BND XIC N9:0/4 BND OTE N51:45/0 EOR
% Rung: 1 %
SOR XIC B3:3/7 MOV N25:22 N25:21 EOR
% Rung: 2 %
SOR XIC B3:3/8 MOV N25:23 N25:21 EOR
% Rung: 3 %
SOR XIC N9:3/3 MOV N100:14 N25:21 EOR
% Rung: 4 %
SOR XIC B3:1/7 XIC B3:3/7 MOV N25:24 N25:21 EOR
% Rung: 5 %
SOR XIC B3:1/7 XIC B3:3/8 MOV N25:25 N25:21 EOR
% Rung: 6 %
SOR XIC B3:1/8 XIC B3:3/7 MOV N25:26 N25:21 EOR
% Rung: 7 %
SOR MOV N25:26 N25:27 EOR

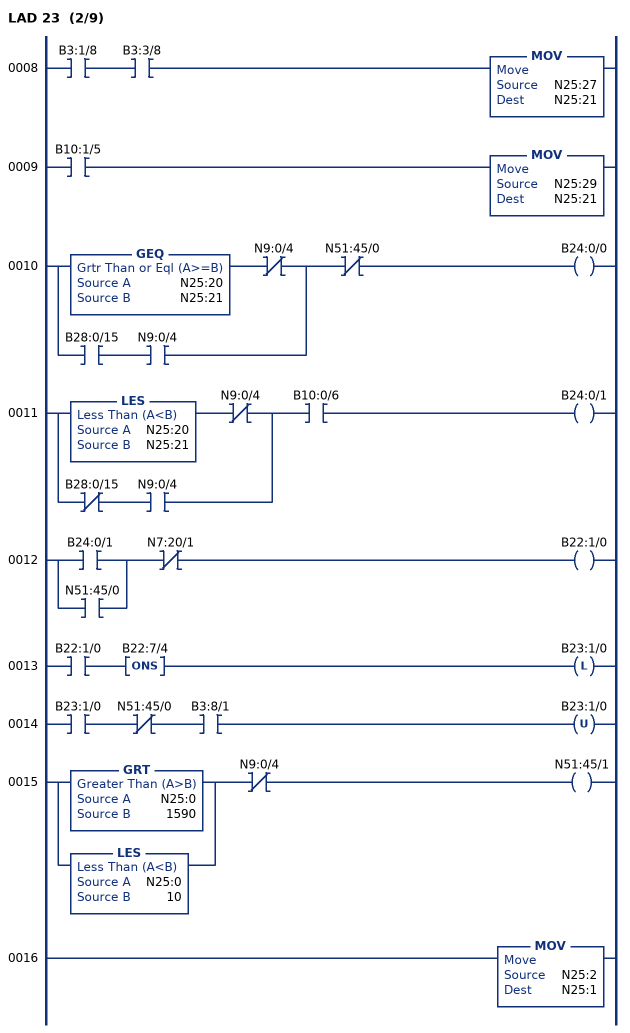
% Rung: 8 %
SOR XIC B3:1/8 XIC B3:3/8 MOV N25:27 N25:21 EOR
% Rung: 9 %
SOR XIC B10:1/5 MOV N25:29 N25:21 EOR
% Rung: 10 %
SOR BST GEQ N25:20 N25:21 XIO N9:0/4 NXB XIC B28:0/15 XIC N9:0/4 BND XIO N51:45/0 OTE B24:0/0 EOR
% Rung: 11 %
SOR BST LES N25:20 N25:21 XIO N9:0/4 NXB XIO B28:0/15 XIC N9:0/4 BND XIC B10:0/6 OTE B24:0/1 EOR
% Rung: 12 %
SOR BST XIC B24:0/1 NXB XIC N51:45/0 BND XIO N7:20/1 OTE B22:1/0 EOR
% Rung: 13 %
SOR XIC B22:1/0 OSR B22:7/4 OTL B23:1/0 EOR
% Rung: 14 %
SOR XIC B23:1/0 XIO N51:45/0 XIC B3:8/1 OTU B23:1/0 EOR
% Rung: 15 %
SOR BST GRT N25:0 1590 NXB LES N25:0 10 BND XIO N9:0/4 OTE N51:45/1 EOR
% Rung: 16 %
SOR MOV N25:2 N25:1 EOR

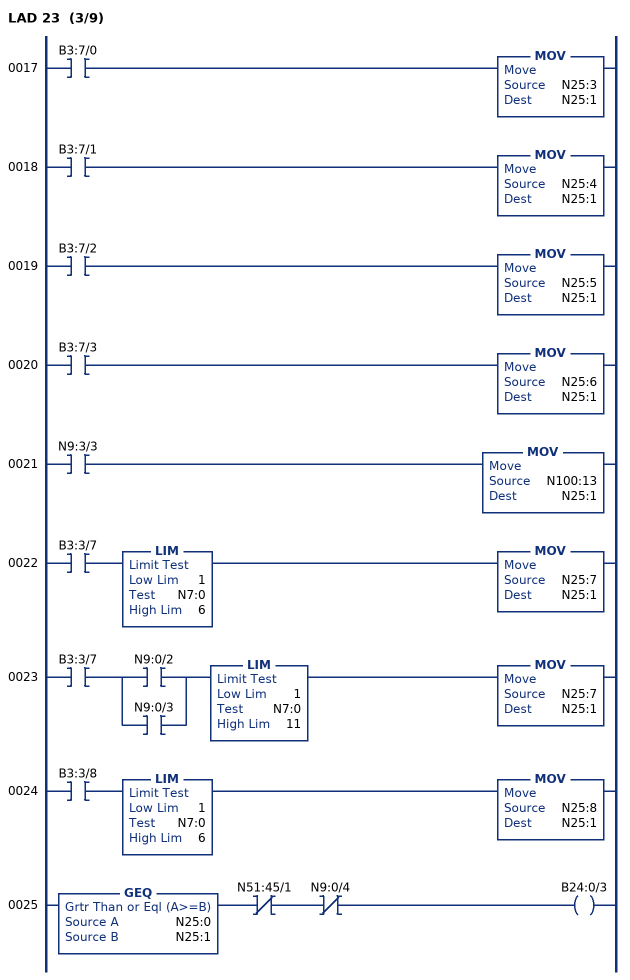
% Rung: 17 %
SOR XIC B3:7/0 MOV N25:3 N25:1 EOR
% Rung: 18 %
SOR XIC B3:7/1 MOV N25:4 N25:1 EOR
% Rung: 19 %
SOR XIC B3:7/2 MOV N25:5 N25:1 EOR
% Rung: 20 %
SOR XIC B3:7/3 MOV N25:6 N25:1 EOR
% Rung: 21 %
SOR XIC N9:3/3 MOV N100:13 N25:1 EOR
% Rung: 22 %
SOR XIC B3:3/7 LIM 1 N7:0 6 MOV N25:7 N25:1 EOR
% Rung: 23 %
SOR XIC B3:3/7 BST XIC N9:0/2 NXB XIC N9:0/3 BND LIM 1 N7:0 11 MOV N25:7 N25:1 EOR
% Rung: 24 %
SOR XIC B3:3/8 LIM 1 N7:0 6 MOV N25:8 N25:1 EOR
% Rung: 25 %
SOR GEQ N25:0 N25:1 XIO N51:45/1 XIO N9:0/4 OTE B24:0/3 EOR

